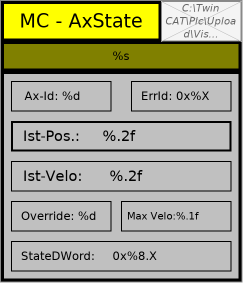
VISUALIZATION MC_AxesInfo  // 243x283
VAR_IN_OUT
	m_Input_Instance : None;
END_VAR
    Group (1,1 238x278)
        Rectangle (0,70 240x210)
        RoundedRectangle (10,120 220x30), "Ist-Pos.: %.2f", text variable: Global_Var_AxisInterface.stAxis[m_Input_Instance].NcToPlc.ActPos
        RoundedRectangle (10,160 220x30), "Ist-Velo: %.2f", text variable: Global_Var_AxisInterface.stAxis[m_Input_Instance].NcToPlc.ActVelo
        RoundedRectangle (130,80 100x30), "ErrId: 0x%X", text variable: Global_Var_AxisInterface.stAxis[m_Input_Instance].NcToPlc.ErrorCode, colour toggle: Global_Var_AxisInterface.stAxis[m_Input_Instance].NcToPlc.ErrorCode <> 0
        RoundedRectangle (10,80 100x30), "Ax-Id: %d", text variable: Global_Var_AxisInterface.stAxis[m_Input_Instance].NcToPlc.AxisId
            toggle Global_Var_AxisInterface.stAxesfunctions[m_Input_Instance].bMcPower
        Rectangle (0,0 160x40), "MC - AxState"
        Rectangle (0,40 240x30), "%s", text variable: m_Input_Instance_Str
        Image (160,0 80x40), image: C:\TwinCAT\Plc\Upload\VisuBmp\\BECKHOFFLOGOKLEIN.BMP
        RoundedRectangle (10,240 220x30), "StateDWord: 0x%8.X", text variable: Global_Var_AxisInterface.stAxis[m_Input_Instance].NcToPlc.StateDWord
        RoundedRectangle (10,200 100x30), "Override: %d", text variable: Global_Var_AxisInterface.stAxis[m_Input_Instance].PlcToNc.Override / 10000
        RoundedRectangle (120,200 110x30), "Max Velo:%.1f", text variable: Global_Var_AxisInterface.stAxesfunctions[m_Input_Instance].NcMaxVelo
END_VISUALIZATION

(* stored: Version 1.1.0.1, ProductVersion 3.1.4024.11
   Visu MC_AxesInfo: Id {4f1a00c3-c1ac-4bb2-ba87-09d007cc39ce} *)
